TYPE M3TargetStates :
(
	NO_TARGET_GIVEN := 0,
	KNOWN_POSITION := 1,
	NEW_POSITION := 2
);
END_TYPE

(* stored: Version 1.1.0.1, ProductVersion 3.1.4019.2
   DUT M3TargetStates: Id {378c64db-1756-4ab7-a72b-4ca100c0f8a3} *)
